TYPE ST_2 :
STRUCT
	bBool : BOOL;
END_STRUCT
END_TYPE

(* stored: Version 1.1.0.1, ProductVersion 3.1.4024.12
   DUT ST_2: Id {dcd9326c-a5b2-4216-9e9f-b0ce42de8354} *)
